PROGRAM Group_01_Function_Blocks
VAR
END_VAR

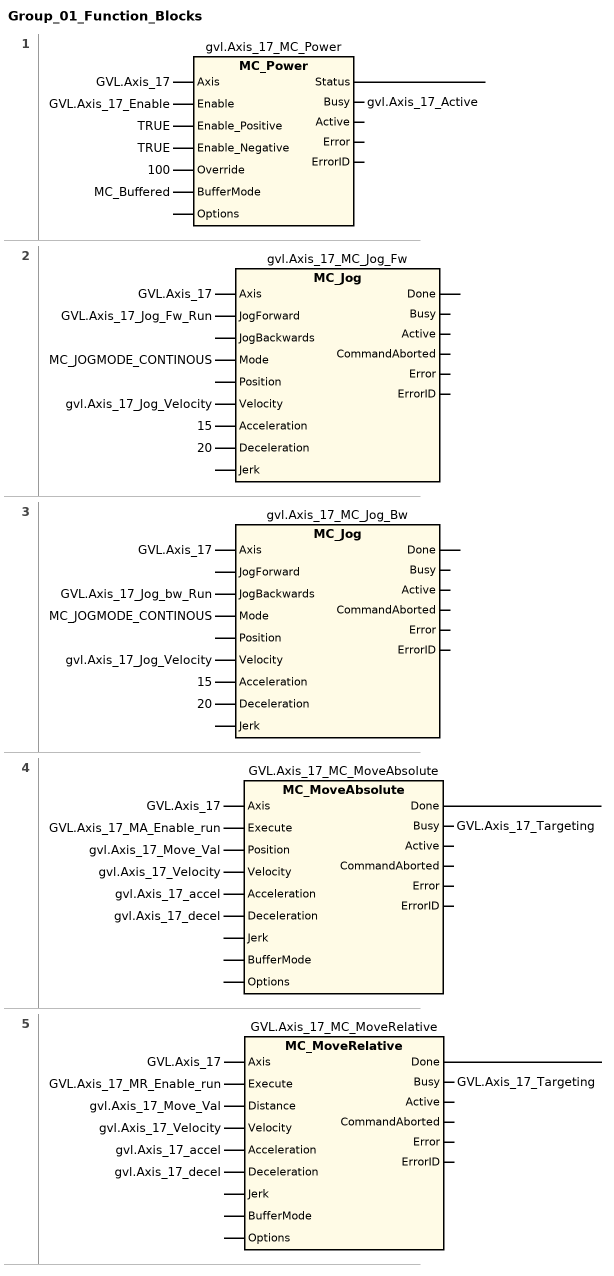
// NETWORK 1
gvl.Axis_17_MC_Power(
    Axis := GVL.Axis_17,
    Enable := GVL.Axis_17_Enable,
    Enable_Positive := TRUE,
    Enable_Negative := TRUE,
    Override := 100,
    BufferMode := MC_Buffered,
    Busy => gvl.Axis_17_Active); // MC_Power

// NETWORK 2
gvl.Axis_17_MC_Jog_Fw(
    Axis := GVL.Axis_17,
    JogForward := GVL.Axis_17_Jog_Fw_Run,
    Mode := MC_JOGMODE_CONTINOUS,
    Velocity := gvl.Axis_17_Jog_Velocity,
    Acceleration := 15,
    Deceleration := 20); // MC_Jog

// NETWORK 3
gvl.Axis_17_MC_Jog_Bw(
    Axis := GVL.Axis_17,
    JogBackwards := GVL.Axis_17_Jog_bw_Run,
    Mode := MC_JOGMODE_CONTINOUS,
    Velocity := gvl.Axis_17_Jog_Velocity,
    Acceleration := 15,
    Deceleration := 20); // MC_Jog

// NETWORK 4
GVL.Axis_17_MC_MoveAbsolute(
    Axis := GVL.Axis_17,
    Execute := GVL.Axis_17_MA_Enable_run,
    Position := gvl.Axis_17_Move_Val,
    Velocity := gvl.Axis_17_Velocity,
    Acceleration := gvl.Axis_17_accel,
    Deceleration := gvl.Axis_17_decel,
    Busy => GVL.Axis_17_Targeting); // MC_MoveAbsolute

// NETWORK 5
GVL.Axis_17_MC_MoveRelative(
    Axis := GVL.Axis_17,
    Execute := GVL.Axis_17_MR_Enable_run,
    Distance := gvl.Axis_17_Move_Val,
    Velocity := gvl.Axis_17_Velocity,
    Acceleration := gvl.Axis_17_accel,
    Deceleration := gvl.Axis_17_decel,
    Busy => GVL.Axis_17_Targeting); // MC_MoveRelative

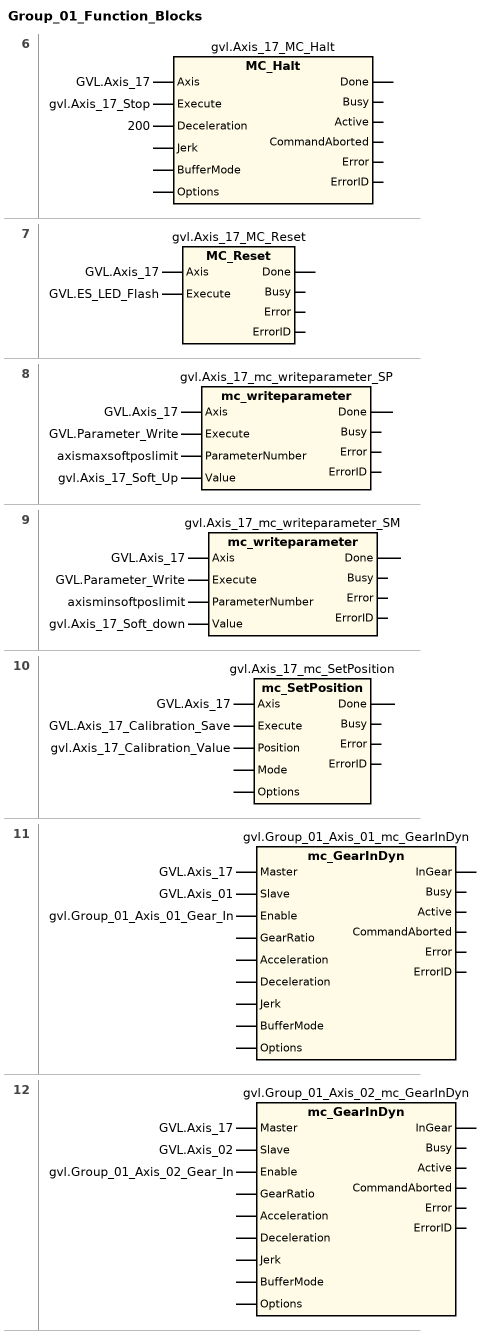
// NETWORK 6
gvl.Axis_17_MC_Halt(Axis := GVL.Axis_17, Execute := gvl.Axis_17_Stop, Deceleration := 200); // MC_Halt

// NETWORK 7
gvl.Axis_17_MC_Reset(Axis := GVL.Axis_17, Execute := GVL.ES_LED_Flash); // MC_Reset

// NETWORK 8
gvl.Axis_17_mc_writeparameter_SP(
    Axis := GVL.Axis_17,
    Execute := GVL.Parameter_Write,
    ParameterNumber := axismaxsoftposlimit,
    Value := gvl.Axis_17_Soft_Up); // mc_writeparameter

// NETWORK 9
gvl.Axis_17_mc_writeparameter_SM(
    Axis := GVL.Axis_17,
    Execute := GVL.Parameter_Write,
    ParameterNumber := axisminsoftposlimit,
    Value := gvl.Axis_17_Soft_down); // mc_writeparameter

// NETWORK 10
gvl.Axis_17_mc_SetPosition(
    Axis := GVL.Axis_17,
    Execute := GVL.Axis_17_Calibration_Save,
    Position := gvl.Axis_17_Calibration_Value); // mc_SetPosition

// NETWORK 11
gvl.Group_01_Axis_01_mc_GearInDyn(
    Master := GVL.Axis_17,
    Slave := GVL.Axis_01,
    Enable := gvl.Group_01_Axis_01_Gear_In); // mc_GearInDyn

// NETWORK 12
gvl.Group_01_Axis_02_mc_GearInDyn(
    Master := GVL.Axis_17,
    Slave := GVL.Axis_02,
    Enable := gvl.Group_01_Axis_02_Gear_In); // mc_GearInDyn

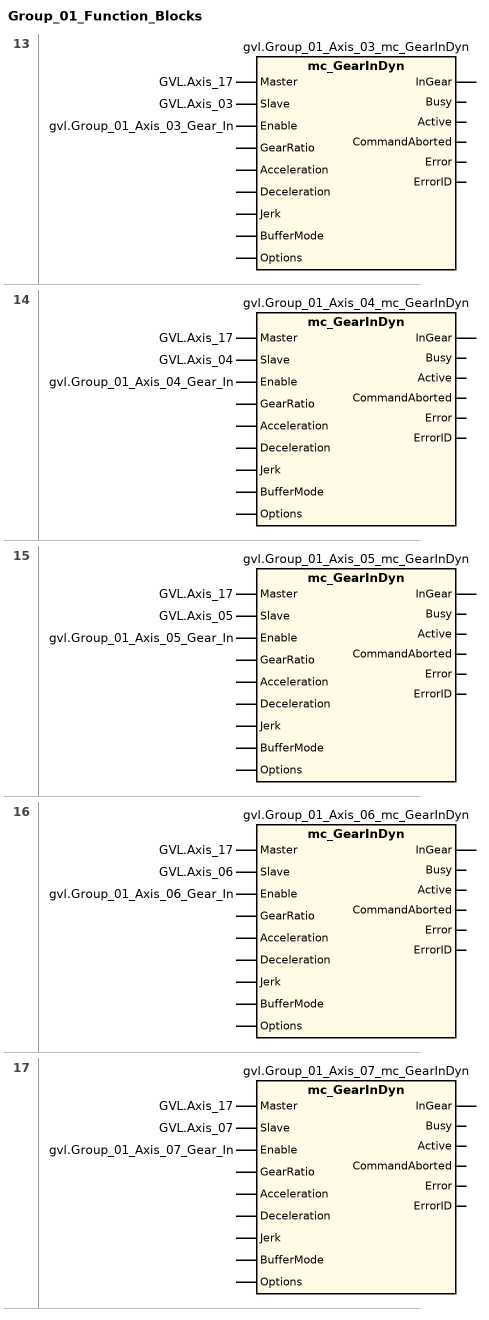
// NETWORK 13
gvl.Group_01_Axis_03_mc_GearInDyn(
    Master := GVL.Axis_17,
    Slave := GVL.Axis_03,
    Enable := gvl.Group_01_Axis_03_Gear_In); // mc_GearInDyn

// NETWORK 14
gvl.Group_01_Axis_04_mc_GearInDyn(
    Master := GVL.Axis_17,
    Slave := GVL.Axis_04,
    Enable := gvl.Group_01_Axis_04_Gear_In); // mc_GearInDyn

// NETWORK 15
gvl.Group_01_Axis_05_mc_GearInDyn(
    Master := GVL.Axis_17,
    Slave := GVL.Axis_05,
    Enable := gvl.Group_01_Axis_05_Gear_In); // mc_GearInDyn

// NETWORK 16
gvl.Group_01_Axis_06_mc_GearInDyn(
    Master := GVL.Axis_17,
    Slave := GVL.Axis_06,
    Enable := gvl.Group_01_Axis_06_Gear_In); // mc_GearInDyn

// NETWORK 17
gvl.Group_01_Axis_07_mc_GearInDyn(
    Master := GVL.Axis_17,
    Slave := GVL.Axis_07,
    Enable := gvl.Group_01_Axis_07_Gear_In); // mc_GearInDyn

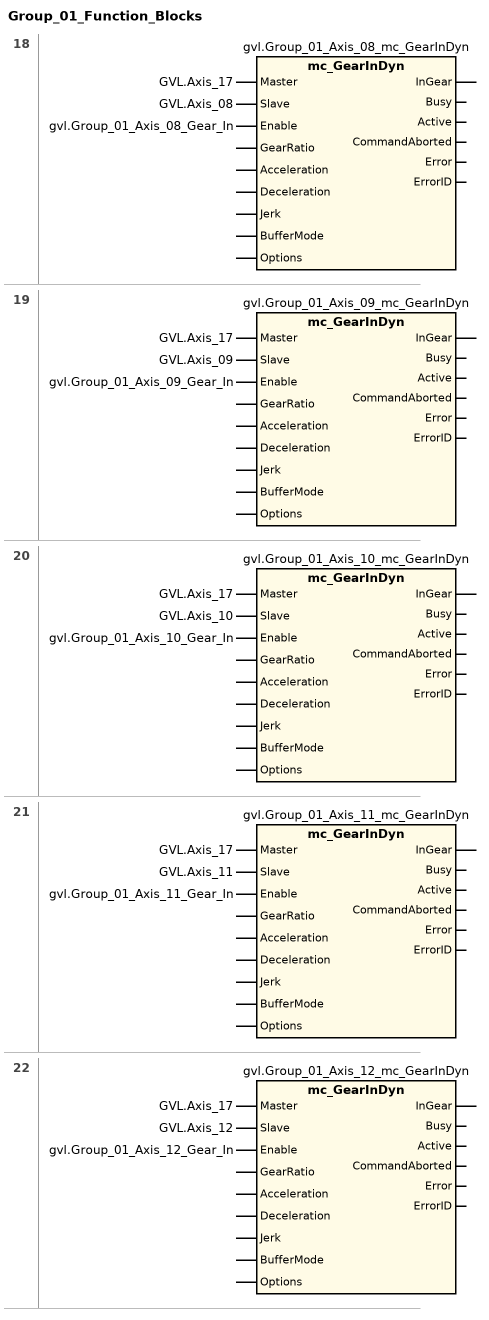
// NETWORK 18
gvl.Group_01_Axis_08_mc_GearInDyn(
    Master := GVL.Axis_17,
    Slave := GVL.Axis_08,
    Enable := gvl.Group_01_Axis_08_Gear_In); // mc_GearInDyn

// NETWORK 19
gvl.Group_01_Axis_09_mc_GearInDyn(
    Master := GVL.Axis_17,
    Slave := GVL.Axis_09,
    Enable := gvl.Group_01_Axis_09_Gear_In); // mc_GearInDyn

// NETWORK 20
gvl.Group_01_Axis_10_mc_GearInDyn(
    Master := GVL.Axis_17,
    Slave := GVL.Axis_10,
    Enable := gvl.Group_01_Axis_10_Gear_In); // mc_GearInDyn

// NETWORK 21
gvl.Group_01_Axis_11_mc_GearInDyn(
    Master := GVL.Axis_17,
    Slave := GVL.Axis_11,
    Enable := gvl.Group_01_Axis_11_Gear_In); // mc_GearInDyn

// NETWORK 22
gvl.Group_01_Axis_12_mc_GearInDyn(
    Master := GVL.Axis_17,
    Slave := GVL.Axis_12,
    Enable := gvl.Group_01_Axis_12_Gear_In); // mc_GearInDyn

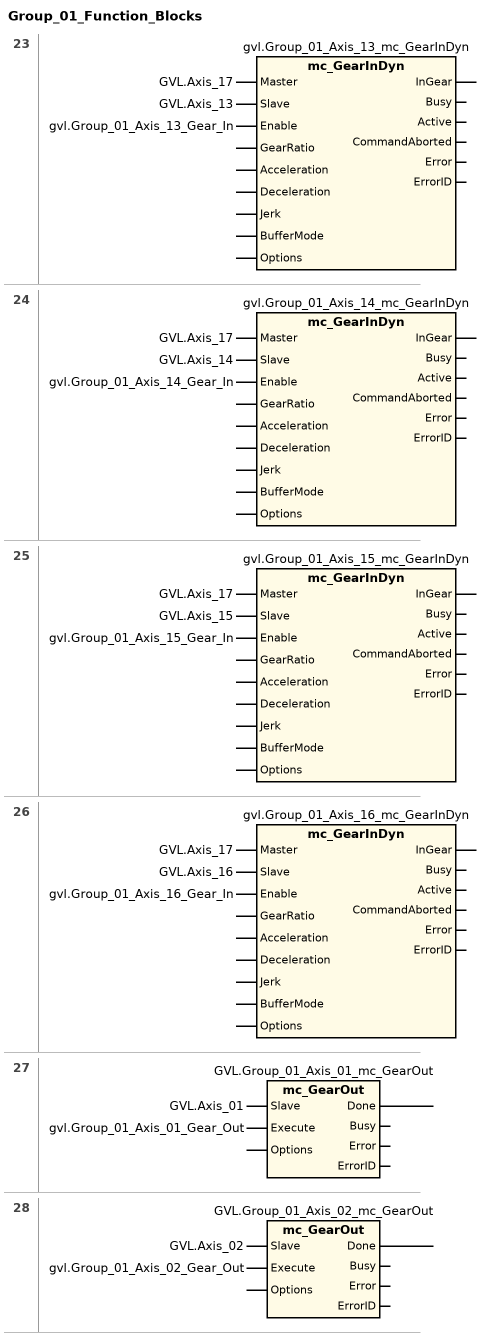
// NETWORK 23
gvl.Group_01_Axis_13_mc_GearInDyn(
    Master := GVL.Axis_17,
    Slave := GVL.Axis_13,
    Enable := gvl.Group_01_Axis_13_Gear_In); // mc_GearInDyn

// NETWORK 24
gvl.Group_01_Axis_14_mc_GearInDyn(
    Master := GVL.Axis_17,
    Slave := GVL.Axis_14,
    Enable := gvl.Group_01_Axis_14_Gear_In); // mc_GearInDyn

// NETWORK 25
gvl.Group_01_Axis_15_mc_GearInDyn(
    Master := GVL.Axis_17,
    Slave := GVL.Axis_15,
    Enable := gvl.Group_01_Axis_15_Gear_In); // mc_GearInDyn

// NETWORK 26
gvl.Group_01_Axis_16_mc_GearInDyn(
    Master := GVL.Axis_17,
    Slave := GVL.Axis_16,
    Enable := gvl.Group_01_Axis_16_Gear_In); // mc_GearInDyn

// NETWORK 27
GVL.Group_01_Axis_01_mc_GearOut(Slave := GVL.Axis_01, Execute := gvl.Group_01_Axis_01_Gear_Out); // mc_GearOut

// NETWORK 28
GVL.Group_01_Axis_02_mc_GearOut(Slave := GVL.Axis_02, Execute := gvl.Group_01_Axis_02_Gear_Out); // mc_GearOut

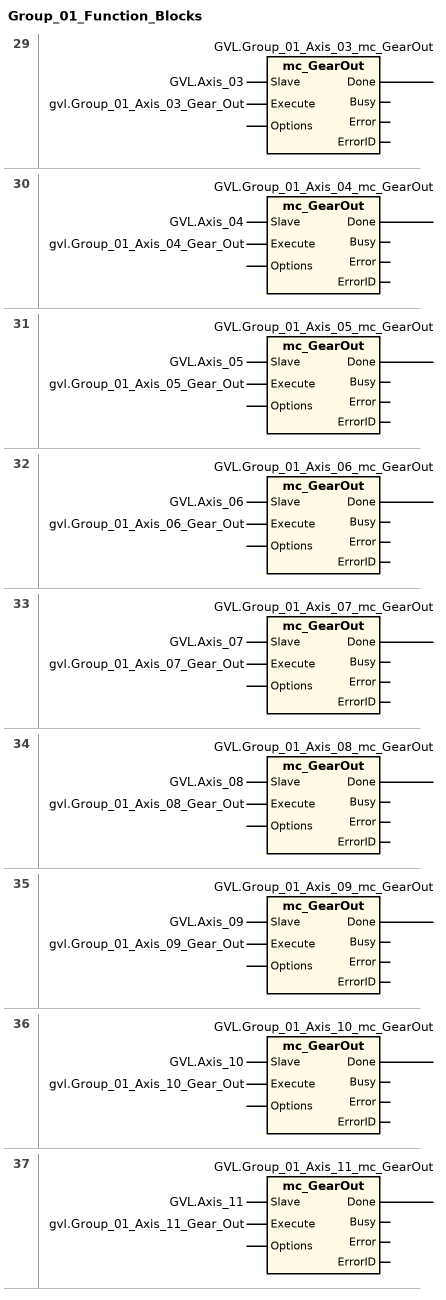
// NETWORK 29
GVL.Group_01_Axis_03_mc_GearOut(Slave := GVL.Axis_03, Execute := gvl.Group_01_Axis_03_Gear_Out); // mc_GearOut

// NETWORK 30
GVL.Group_01_Axis_04_mc_GearOut(Slave := GVL.Axis_04, Execute := gvl.Group_01_Axis_04_Gear_Out); // mc_GearOut

// NETWORK 31
GVL.Group_01_Axis_05_mc_GearOut(Slave := GVL.Axis_05, Execute := gvl.Group_01_Axis_05_Gear_Out); // mc_GearOut

// NETWORK 32
GVL.Group_01_Axis_06_mc_GearOut(Slave := GVL.Axis_06, Execute := gvl.Group_01_Axis_06_Gear_Out); // mc_GearOut

// NETWORK 33
GVL.Group_01_Axis_07_mc_GearOut(Slave := GVL.Axis_07, Execute := gvl.Group_01_Axis_07_Gear_Out); // mc_GearOut

// NETWORK 34
GVL.Group_01_Axis_08_mc_GearOut(Slave := GVL.Axis_08, Execute := gvl.Group_01_Axis_08_Gear_Out); // mc_GearOut

// NETWORK 35
GVL.Group_01_Axis_09_mc_GearOut(Slave := GVL.Axis_09, Execute := gvl.Group_01_Axis_09_Gear_Out); // mc_GearOut

// NETWORK 36
GVL.Group_01_Axis_10_mc_GearOut(Slave := GVL.Axis_10, Execute := gvl.Group_01_Axis_10_Gear_Out); // mc_GearOut

// NETWORK 37
GVL.Group_01_Axis_11_mc_GearOut(Slave := GVL.Axis_11, Execute := gvl.Group_01_Axis_11_Gear_Out); // mc_GearOut

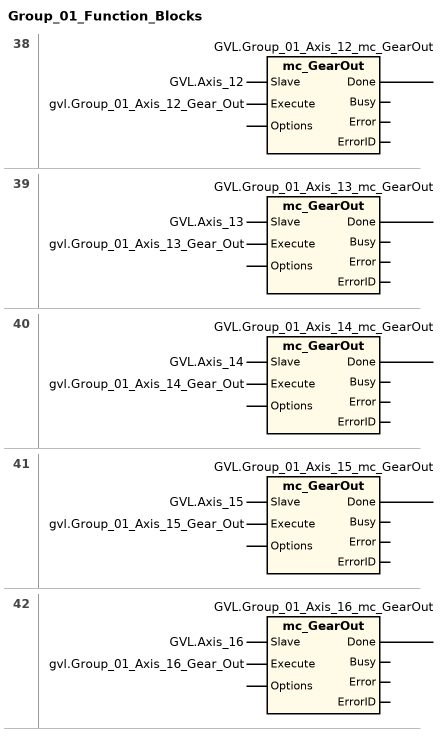
// NETWORK 38
GVL.Group_01_Axis_12_mc_GearOut(Slave := GVL.Axis_12, Execute := gvl.Group_01_Axis_12_Gear_Out); // mc_GearOut

// NETWORK 39
GVL.Group_01_Axis_13_mc_GearOut(Slave := GVL.Axis_13, Execute := gvl.Group_01_Axis_13_Gear_Out); // mc_GearOut

// NETWORK 40
GVL.Group_01_Axis_14_mc_GearOut(Slave := GVL.Axis_14, Execute := gvl.Group_01_Axis_14_Gear_Out); // mc_GearOut

// NETWORK 41
GVL.Group_01_Axis_15_mc_GearOut(Slave := GVL.Axis_15, Execute := gvl.Group_01_Axis_15_Gear_Out); // mc_GearOut

// NETWORK 42
GVL.Group_01_Axis_16_mc_GearOut(Slave := GVL.Axis_16, Execute := gvl.Group_01_Axis_16_Gear_Out); // mc_GearOut

END_PROGRAM

(* stored: Version 1.1.0.1, ProductVersion 3.1.4022.12
   POU Group_01_Function_Blocks: Id {b88d6449-08ac-4c82-9006-5b6891f8b465}, SpecialFunc None *)
